Staubli VAL3: onF6Event.pgx

program onF6Event()
  local string l_sMessage
  local bool l_bYes
  local num l_nSize
  local num l_nFound
  local string l_sEvent
  local string l_sButton[2]
  local num l_nItem
begin
end
